KUKA KRL program: up24.src, up24.dat

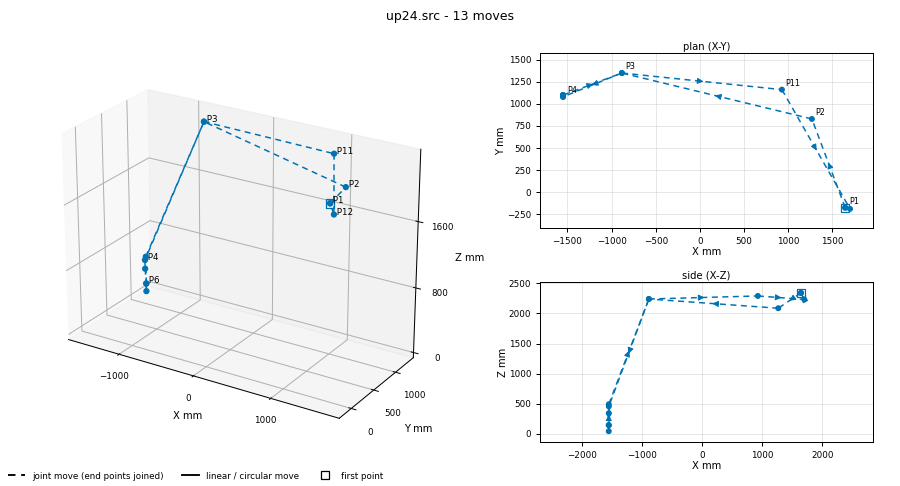
[picture p0: tool path of up24.src, 13 of 13 moves have a stored position in this frame; points joined in program order, loops and branches not executed]
--- up24.src ---
&ACCESS RV7
&REL 180
&COMMENT VW380 Ablegen AFO 115440
&PARAM DISKPATH = KRC:\R1\UPs
&PARAM TEMPLATE = C:\KRC\Roboter\Template\upvorgabe
&PARAM TPVW_VERSION = 8.1.8
&PARAM EDITMASK = Up999[1-999]
DEF UP24()
   ; FOLD UP Anfang;%{SE} %MKUKATPVW
   SPS_N=-1
   SPS_FERTIG=FALSE
   IF NOT CALLBYSELECT THEN
      INTERRUPT DECL 10 WHEN $CYCFLAG[254]==FALSE DO VW(#FB_STOP,TRUE)
      INTERRUPT ON 10
      INT10=TRUE
      VW_USR_R (#USR_INIT)
   ENDIF
   VW(#VW_INIT_UP,TRUE)
   ; ENDFOLD
   ;FOLD -- K2TUHR115425R01 -- ;%{PSE}%MKUKATPVW,%CVW_COM,%VCOMMENT,%P 1:Comment:, 2:K2TUHR115425R01
      ;FOLD {H}
         M_COMMENT("K2TUHR115425R01")
      ;ENDFOLD
   ;ENDFOLD
   ;FOLD -- VW370 Ablegen AFO 115440 -- ;%{PSE}%MKUKATPVW,%CVW_COM,%VCOMMENT,%P 1:Comment:, 2:VW370 Ablegen AFO 115440
      ;FOLD {H}
         M_COMMENT("VW370 Ablegen AFO 115440")
      ;ENDFOLD
   ;ENDFOLD
   ;FOLD -- Verriegelung (E43) an Rob 5440R01 EIN -- ;%{PSE}%MKUKATPVW,%CVW_COM,%VCOMMENT,%P 1:Comment:, 2:Verriegelung (E43) an Rob 5440R01 EIN
      ;FOLD {H}
         M_COMMENT("Verriegelung (E43) an Rob 5440R01 EIN")
      ;ENDFOLD
   ;ENDFOLD
   ;FOLD -- Verriegelung (E45) an Rob 5430R01 EIN -- ;%{PSE}%MKUKATPVW,%CVW_COM,%VCOMMENT,%P 1:Comment:, 2:Verriegelung (E45) an Rob 5430R01 EIN
      ;FOLD {H}
         M_COMMENT("Verriegelung (E45) an Rob 5430R01 EIN")
      ;ENDFOLD
   ;ENDFOLD
   ;FOLD -- Verriegelung (E54) an Rob 5450R01 EIN -- ;%{PSE}%MKUKATPVW,%CVW_COM,%VCOMMENT,%P 1:Comment:, 2:Verriegelung (E54) an Rob 5450R01 EIN
      ;FOLD {H}
         M_COMMENT("Verriegelung (E54) an Rob 5450R01 EIN")
      ;ENDFOLD
   ;ENDFOLD
   ;FOLD -- Profilfrei AFO 115440 AUS -- ;%{PSE}%MKUKATPVW,%CVW_COM,%VCOMMENT,%P 1:Comment:, 2:Profilfrei AFO 115440 AUS
      ;FOLD {H}
         M_COMMENT("Profilfrei AFO 115440 AUS")
      ;ENDFOLD
   ;ENDFOLD
   ;FOLD -- Profilfrei DT 115440 AUS -- ;%{PSE}%MKUKATPVW,%CVW_COM,%VCOMMENT,%P 1:Comment:, 2:Profilfrei DT 115440 AUS
      ;FOLD {H}
         M_COMMENT("Profilfrei DT 115440 AUS")
      ;ENDFOLD
   ;ENDFOLD
   ;FOLD -- Wartungsbereich -- ;%{PSE}%MKUKATPVW,%CVW_COM,%VCOMMENT,%P 1:Comment:, 2:Wartungsbereich
      ;FOLD {H}
         M_COMMENT("Wartungsbereich")
      ;ENDFOLD
   ;ENDFOLD
;FOLD PTP VB=100% VE=0% ACC=100% RobWzg=12 Base=0 SPSTrig=0[1/100s] P;%{P}%MKUKATPVW,%CMOVE8,%VPTP,%P 1:1, 2: VB=, 3:100, 4:%, 5: VE=, 6:0, 7:%, 8: ACC=, 9:100, 10:%, 11: RobWzg=, 12:12, 13: Base=, 14:0, 15: SPSTrig=, 16:0, 17:[1/100s], 18: P, 19:1, 20:-1, 21:1
;FOLD 1: FB PSPS = EIN;%{SE}%MKUKATPVW %CVW_SPS %VFBPSPS %P 2:FB PSPS = EIN,3: FBPSPS
;ENDFOLD
;FOLD 2: A23 = AUS;%{SE}%MKUKATPVW %CVW_SPS %VBOASG %P 2:A23 = AUS,3: BOASG
;ENDFOLD
;FOLD 3: t3 ( EIN ) = 0[1/10Sek];%{SE}%MKUKATPVW %CVW_SPS %VTASG %P 2:t3 ( EIN ) = 0[1/10Sek],3: TASG
;ENDFOLD
;FOLD 4: SPSMAKRO50 = EIN;%{SE}%MKUKATPVW %CVW_SPS %VMAKRO %P 2:SPSMAKRO50 = EIN,3: MAKRO
;ENDFOLD
;FOLD 5: SPSMAKRO53 = EIN;%{SE}%MKUKATPVW %CVW_SPS %VMAKRO %P 2:SPSMAKRO53 = EIN,3: MAKRO
;ENDFOLD
;FOLD 6: A42 = EIN;%{SE}%MKUKATPVW %CVW_SPS %VBOASG %P 2:A42 = EIN,3: BOASG
;ENDFOLD
;FOLD 7: A43 = EIN;%{SE}%MKUKATPVW %CVW_SPS %VBOASG %P 2:A43 = EIN,3: BOASG
;ENDFOLD
;FOLD 8: A44 = EIN;%{SE}%MKUKATPVW %CVW_SPS %VBOASG %P 2:A44 = EIN,3: BOASG
;ENDFOLD
;FOLD 9: A45 = EIN;%{SE}%MKUKATPVW %CVW_SPS %VBOASG %P 2:A45 = EIN,3: BOASG
;ENDFOLD
;FOLD 10: A47 = EIN;%{SE}%MKUKATPVW %CVW_SPS %VBOASG %P 2:A47 = EIN,3: BOASG
;ENDFOLD
;FOLD 11: A49 = EIN;%{SE}%MKUKATPVW %CVW_SPS %VBOASG %P 2:A49 = EIN,3: BOASG
;ENDFOLD
;FOLD 12: A50 = EIN;%{SE}%MKUKATPVW %CVW_SPS %VBOASG %P 2:A50 = EIN,3: BOASG
;ENDFOLD
;FOLD 13: A52 = EIN;%{SE}%MKUKATPVW %CVW_SPS %VBOASG %P 2:A52 = EIN,3: BOASG
;ENDFOLD
;FOLD 14: A54 = EIN;%{SE}%MKUKATPVW %CVW_SPS %VBOASG %P 2:A54 = EIN,3: BOASG
;ENDFOLD
;FOLD 15: A75 = EIN;%{SE}%MKUKATPVW %CVW_SPS %VBOASG %P 2:A75 = EIN,3: BOASG
;ENDFOLD
;FOLD 16: A76 = EIN;%{SE}%MKUKATPVW %CVW_SPS %VBOASG %P 2:A76 = EIN,3: BOASG
;ENDFOLD
;FOLD 17: A79 = EIN;%{SE}%MKUKATPVW %CVW_SPS %VBOASG %P 2:A79 = EIN,3: BOASG
;ENDFOLD
;FOLD 18: A80 = EIN;%{SE}%MKUKATPVW %CVW_SPS %VBOASG %P 2:A80 = EIN,3: BOASG
;ENDFOLD
;FOLD 19: A18 = EIN;%{SE}%MKUKATPVW %CVW_SPS %VBOASG %P 2:A18 = EIN,3: BOASG
;ENDFOLD
;FOLD 20: WARTE BIS E43 & E45 & E54 & !E59 & E60 & E75 & E76 & (!E18 + E19);%{SE}%MKUKATPVW %CVW_SPS %VWBOASG %P 2:WARTE BIS E43 & E45 & E54 & !E59 & E60 & E75 & E76 & (!E18 + E19),3: WBOASG
;ENDFOLD
;FOLD 21: A18 = AUS;%{SE}%MKUKATPVW %CVW_SPS %VBOASG %P 2:A18 = AUS,3: BOASG
;ENDFOLD
;FOLD 22: F2 = EIN;%{SE}%MKUKATPVW %CVW_SPS %VBOASG %P 2:F2 = EIN,3: BOASG
;ENDFOLD
;FOLD 23: SPSMAKRO343 = EIN;%{SE}%MKUKATPVW %CVW_SPS %VMAKRO %P 2:SPSMAKRO343 = EIN,3: MAKRO
;ENDFOLD
;FOLD 24: WARTE BIS M34;%{SE}%MKUKATPVW %CVW_SPS %VWBOASG %P 2:WARTE BIS M34,3: WBOASG
;ENDFOLD
;FOLD 25: A75 = AUS;%{SE}%MKUKATPVW %CVW_SPS %VBOASG %P 2:A75 = AUS,3: BOASG
;ENDFOLD
;FOLD 26: A76 = AUS;%{SE}%MKUKATPVW %CVW_SPS %VBOASG %P 2:A76 = AUS,3: BOASG
;ENDFOLD
;FOLD 27: A83 = EIN;%{SE}%MKUKATPVW %CVW_SPS %VBOASG %P 2:A83 = EIN,3: BOASG
;ENDFOLD
;FOLD 28: A85 = EIN;%{SE}%MKUKATPVW %CVW_SPS %VBOASG %P 2:A85 = EIN,3: BOASG
;ENDFOLD
;FOLD 29: A94 = EIN;%{SE}%MKUKATPVW %CVW_SPS %VBOASG %P 2:A94 = EIN,3: BOASG
;ENDFOLD
;FOLD 30: SPSMAKRO20 = EIN;%{SE}%MKUKATPVW %CVW_SPS %VMAKRO %P 2:SPSMAKRO20 = EIN,3: MAKRO
;ENDFOLD
;FOLD 31: WARTE BIS E23;%{SE}%MKUKATPVW %CVW_SPS %VWBOASG %P 2:WARTE BIS E23,3: WBOASG
;ENDFOLD
;FOLD 32: A23 = EIN;%{SE}%MKUKATPVW %CVW_SPS %VBOASG %P 2:A23 = EIN,3: BOASG
;ENDFOLD
;FOLD 33: FB PSPS = M1 & M28 & M30 & M32 & M34 & M78 & E60 & E75 & E76;%{SE}%MKUKATPVW %CVW_SPS %VFBPSPS %P 2:FB PSPS = M1 & M28 & M30 & M32 & M34 & M78 & E60 & E75 & E76,3: FBPSPS
;ENDFOLD
;FOLD {H}
VW_MPARA_ACT = P1_D
Act_P1 = P1
Act_P2 = P1
VW(#MPARA,TRUE)
SPS_FERTIG=FALSE
TRIGGER WHEN DISTANCE=1 DELAY=0 DO SPS_TRIG(1) PRIO=-1
PTP P1
$ADVANCE=1
WAIT FOR SPS_FERTIG
;ENDFOLD
;ENDFOLD
   ;FOLD PTP VB=100% VE=100% ACC=100% RobWzg=12 Base=0 SPSTrig=0[1/100s] P ;%{P}%MKUKATPVW,%CMOVE8,%VPTP,%P 1:1, 2: VB=, 3:100, 4:%, 5: VE=, 6:100, 7:%, 8: ACC=, 9:100, 10:%, 11: RobWzg=, 12:12, 13: Base=, 14:0, 15: SPSTrig=, 16:0, 17:[1/100s], 18: P, 19:2, 20:-1, 21:2
      ;FOLD 1: FB PSPS = M1 & M28 & M30 & M32 & M34 & M78 & E60 & E75 & E76 ;%{SE}%MKUKATPVW %CVW_SPS %VFBPSPS %P 2:FB PSPS = M1 & M28 & M30 & M32 & M34 & M78 & E60 & E75 & E76,3:FBPSPS
      ;ENDFOLD
      ;FOLD {H}
         VW_MPARA_ACT=P2_D
         Act_P1 = P2
         Act_P2 = P2
         VW(#MPARA,TRUE)
         SPS_FERTIG=FALSE
         TRIGGER WHEN DISTANCE=1 DELAY=0 DO SPS_TRIG(10002) PRIO=-1
         PTP P2 C_PTP C_VEL
         $ADVANCE=1
      ;ENDFOLD
   ;ENDFOLD
   ;FOLD PTP VB=100% VE=100% ACC=100% RobWzg=12 Base=0 SPSTrig=0[1/100s] P ;%{P}%MKUKATPVW,%CMOVE8,%VPTP,%P 1:1, 2: VB=, 3:100, 4:%, 5: VE=, 6:100, 7:%, 8: ACC=, 9:100, 10:%, 11: RobWzg=, 12:12, 13: Base=, 14:0, 15: SPSTrig=, 16:0, 17:[1/100s], 18: P, 19:3, 20:-1, 21:3
      ;FOLD 1: FB PSPS = M1 & M28 & M30 & M32 & M34 & M78 & E60 & E75 & E76 ;%{SE}%MKUKATPVW %CVW_SPS %VFBPSPS %P 2:FB PSPS = M1 & M28 & M30 & M32 & M34 & M78 & E60 & E75 & E76,3:FBPSPS
      ;ENDFOLD
      ;FOLD {H}
         VW_MPARA_ACT=P3_D
         Act_P1 = P3
         Act_P2 = P3
         VW(#MPARA,TRUE)
         SPS_FERTIG=FALSE
         TRIGGER WHEN DISTANCE=1 DELAY=0 DO SPS_TRIG(10003) PRIO=-1
         PTP P3 C_PTP C_VEL
         $ADVANCE=1
      ;ENDFOLD
   ;ENDFOLD
   ;FOLD PTP VB=100% VE=100% ACC=100% RobWzg=12 Base=0 SPSTrig=0[1/100s] P ;%{P}%MKUKATPVW,%CMOVE8,%VPTP,%P 1:1, 2: VB=, 3:100, 4:%, 5: VE=, 6:100, 7:%, 8: ACC=, 9:100, 10:%, 11: RobWzg=, 12:12, 13: Base=, 14:0, 15: SPSTrig=, 16:0, 17:[1/100s], 18: P, 19:4, 20:-1, 21:4
      ;FOLD 1: FB PSPS = M1 & M28 & M30 & M32 & M34 & M78 & E75 & E76 ;%{SE}%MKUKATPVW %CVW_SPS %VFBPSPS %P 2:FB PSPS = M1 & M28 & M30 & M32 & M34 & M78 & E75 & E76,3:FBPSPS
      ;ENDFOLD
      ;FOLD {H}
         VW_MPARA_ACT=P4_D
         Act_P1 = P4
         Act_P2 = P4
         VW(#MPARA,TRUE)
         SPS_FERTIG=FALSE
         TRIGGER WHEN DISTANCE=1 DELAY=0 DO SPS_TRIG(10004) PRIO=-1
         PTP P4 C_PTP C_VEL
         $ADVANCE=1
      ;ENDFOLD
   ;ENDFOLD
   ;FOLD PTP VB=100% VE=100% ACC=100% RobWzg=12 Base=0 SPSTrig=0[1/100s] P ;%{P}%MKUKATPVW,%CMOVE8,%VPTP,%P 1:1, 2: VB=, 3:100, 4:%, 5: VE=, 6:100, 7:%, 8: ACC=, 9:100, 10:%, 11: RobWzg=, 12:12, 13: Base=, 14:0, 15: SPSTrig=, 16:0, 17:[1/100s], 18: P, 19:5, 20:-1, 21:5
      ;FOLD 1: FB PSPS = M1 & M28 & M30 & M32 & M34 & M78 & E75 & E76 ;%{SE}%MKUKATPVW %CVW_SPS %VFBPSPS %P 2:FB PSPS = M1 & M28 & M30 & M32 & M34 & M78 & E75 & E76,3:FBPSPS
      ;ENDFOLD
      ;FOLD {H}
         VW_MPARA_ACT=P5_D
         Act_P1 = P5
         Act_P2 = P5
         VW(#MPARA,TRUE)
         SPS_FERTIG=FALSE
         TRIGGER WHEN DISTANCE=1 DELAY=0 DO SPS_TRIG(10005) PRIO=-1
         PTP P5 C_PTP C_VEL
         $ADVANCE=1
      ;ENDFOLD
   ;ENDFOLD
   ;FOLD PTP VB=100% VE=10% ACC=100% RobWzg=12 Base=0 SPSTrig=0[1/100s] P ;%{P}%MKUKATPVW,%CMOVE8,%VPTP,%P 1:1, 2: VB=, 3:100, 4:%, 5: VE=, 6:10, 7:%, 8: ACC=, 9:100, 10:%, 11: RobWzg=, 12:12, 13: Base=, 14:0, 15: SPSTrig=, 16:0, 17:[1/100s], 18: P, 19:6, 20:-1, 21:6
      ;FOLD 1: FB PSPS = M1 & M28 & M30 & M32 & M34 & M78 & E75 & E76 ;%{SE}%MKUKATPVW %CVW_SPS %VFBPSPS %P 2:FB PSPS = M1 & M28 & M30 & M32 & M34 & M78 & E75 & E76,3:FBPSPS
      ;ENDFOLD
      ;FOLD {H}
         VW_MPARA_ACT=P6_D
         Act_P1 = P6
         Act_P2 = P6
         VW(#MPARA,TRUE)
         SPS_FERTIG=FALSE
         TRIGGER WHEN DISTANCE=1 DELAY=0 DO SPS_TRIG(10006) PRIO=-1
         PTP P6 C_PTP C_VEL
         $ADVANCE=1
      ;ENDFOLD
   ;ENDFOLD
   ;FOLD -- Bauteil ablegen AFO 115440 -- ;%{PSE}%MKUKATPVW,%CVW_COM,%VCOMMENT,%P 1:Comment:, 2:Bauteil ablegen AFO 115440
      ;FOLD {H}
         M_COMMENT("Bauteil ablegen AFO 115440")
      ;ENDFOLD
   ;ENDFOLD
   ;FOLD -- Greifer auf -- ;%{PSE}%MKUKATPVW,%CVW_COM,%VCOMMENT,%P 1:Comment:, 2:Greifer auf
      ;FOLD {H}
         M_COMMENT("Greifer auf")
      ;ENDFOLD
   ;ENDFOLD
   ;FOLD LIN VB=250[mm/s] VE=0% ACC=100% RobWzg=12 Base=0 SPSTrig=5[1/100s] P ;%{P}%MKUKATPVW,%CMOVE8,%VLIN,%P 1:2, 2: VB=, 3:250, 4:[mm/s], 5: VE=, 6:0, 7:%, 8: ACC=, 9:100, 10:%, 11: RobWzg=, 12:12, 13: Base=, 14:0, 15: SPSTrig=, 16:5, 17:[1/100s], 18: P, 19:7, 20:-1, 21:7
      ;FOLD 1: FB PSPS = EIN ;%{SE}%MKUKATPVW %CVW_SPS %VFBPSPS %P 2:FB PSPS = EIN,3:FBPSPS
      ;ENDFOLD
      ;FOLD 2: A23 = AUS ;%{SE}%MKUKATPVW %CVW_SPS %VBOASG %P 2:A23 = AUS,3:BOASG
      ;ENDFOLD
      ;FOLD 3: A73 = EIN ;%{SE}%MKUKATPVW %CVW_SPS %VBOASG %P 2:A73 = EIN,3:BOASG
      ;ENDFOLD
      ;FOLD 4: WARTE BIS E59 & !E60 ;%{SE}%MKUKATPVW %CVW_SPS %VWBOASG %P 2:WARTE BIS E59 & !E60,3:WBOASG
      ;ENDFOLD
      ;FOLD 5: A74 = EIN ;%{SE}%MKUKATPVW %CVW_SPS %VBOASG %P 2:A74 = EIN,3:BOASG
      ;ENDFOLD
      ;FOLD 6: F1 = EIN ;%{SE}%MKUKATPVW %CVW_SPS %VBOASG %P 2:F1 = EIN,3:BOASG
      ;ENDFOLD
      ;FOLD 7: SPSMAKRO342 = EIN ;%{SE}%MKUKATPVW %CVW_SPS %VMAKRO %P 2:SPSMAKRO342 = EIN,3:MAKRO
      ;ENDFOLD
      ;FOLD 8: SPSMAKRO340 = EIN ;%{SE}%MKUKATPVW %CVW_SPS %VMAKRO %P 2:SPSMAKRO340 = EIN,3:MAKRO
      ;ENDFOLD
      ;FOLD 9: WARTE BIS M31 & M34 ;%{SE}%MKUKATPVW %CVW_SPS %VWBOASG %P 2:WARTE BIS M31 & M34,3:WBOASG
      ;ENDFOLD
      ;FOLD 10: SPSMAKRO4 = EIN ;%{SE}%MKUKATPVW %CVW_SPS %VMAKRO %P 2:SPSMAKRO4 = EIN,3:MAKRO
      ;ENDFOLD
      ;FOLD 11: WARTE BIS E74 ;%{SE}%MKUKATPVW %CVW_SPS %VWBOASG %P 2:WARTE BIS E74,3:WBOASG
      ;ENDFOLD
      ;FOLD 12: A73 = AUS ;%{SE}%MKUKATPVW %CVW_SPS %VBOASG %P 2:A73 = AUS,3:BOASG
      ;ENDFOLD
      ;FOLD 13: A74 = AUS ;%{SE}%MKUKATPVW %CVW_SPS %VBOASG %P 2:A74 = AUS,3:BOASG
      ;ENDFOLD
      ;FOLD 14: WARTE BIS E23 ;%{SE}%MKUKATPVW %CVW_SPS %VWBOASG %P 2:WARTE BIS E23,3:WBOASG
      ;ENDFOLD
      ;FOLD 15: A23 = EIN ;%{SE}%MKUKATPVW %CVW_SPS %VBOASG %P 2:A23 = EIN,3:BOASG
      ;ENDFOLD
      ;FOLD 16: FB PSPS = M28 & M30 & M31 & M34 & M78 & E59 & E74 & E76 ;%{SE}%MKUKATPVW %CVW_SPS %VFBPSPS %P 2:FB PSPS = M28 & M30 & M31 & M34 & M78 & E59 & E74 & E76,3:FBPSPS
      ;ENDFOLD
      ;FOLD {H}
         VW_MPARA_ACT=P7_D
         Act_P1 = P7
         Act_P2 = P7
         VW(#MPARA,TRUE)
         SPS_FERTIG=FALSE
         TRIGGER WHEN DISTANCE=1 DELAY=-50 DO SPS_TRIG(7) PRIO=-1
         LIN P7
         $ADVANCE=1
         WAIT FOR SPS_FERTIG
      ;ENDFOLD
   ;ENDFOLD
   ;FOLD LIN VB=300[mm/s] VE=100% ACC=100% RobWzg=12 Base=0 SPSTrig=0[1/100s] P ;%{P}%MKUKATPVW,%CMOVE8,%VLIN,%P 1:2, 2: VB=, 3:300, 4:[mm/s], 5: VE=, 6:100, 7:%, 8: ACC=, 9:100, 10:%, 11: RobWzg=, 12:12, 13: Base=, 14:0, 15: SPSTrig=, 16:0, 17:[1/100s], 18: P, 19:8, 20:-1, 21:8
      ;FOLD 1: FB PSPS = M13 & M28 & M30 & M31 & M34 & M78 & E59 & E74 & E76 ;%{SE}%MKUKATPVW %CVW_SPS %VFBPSPS %P 2:FB PSPS = M13 & M28 & M30 & M31 & M34 & M78 & E59 & E74 & E76,3:FBPSPS
      ;ENDFOLD
      ;FOLD {H}
         VW_MPARA_ACT=P8_D
         Act_P1 = P8
         Act_P2 = P8
         VW(#MPARA,TRUE)
         SPS_FERTIG=FALSE
         TRIGGER WHEN DISTANCE=1 DELAY=0 DO SPS_TRIG(10008) PRIO=-1
         LIN P8 C_VEL
         $ADVANCE=1
      ;ENDFOLD
   ;ENDFOLD
   ;FOLD PTP VB=100% VE=100% ACC=100% RobWzg=12 Base=0 SPSTrig=0[1/100s] P ;%{P}%MKUKATPVW,%CMOVE8,%VPTP,%P 1:1, 2: VB=, 3:100, 4:%, 5: VE=, 6:100, 7:%, 8: ACC=, 9:100, 10:%, 11: RobWzg=, 12:12, 13: Base=, 14:0, 15: SPSTrig=, 16:0, 17:[1/100s], 18: P, 19:9, 20:-1, 21:9
      ;FOLD 1: FB PSPS = M13 & M28 & M30 & M31 & M34 & M78 & E59 & E74 & E76 ;%{SE}%MKUKATPVW %CVW_SPS %VFBPSPS %P 2:FB PSPS = M13 & M28 & M30 & M31 & M34 & M78 & E59 & E74 & E76,3:FBPSPS
      ;ENDFOLD
      ;FOLD {H}
         VW_MPARA_ACT=P9_D
         Act_P1 = P9
         Act_P2 = P9
         VW(#MPARA,TRUE)
         SPS_FERTIG=FALSE
         TRIGGER WHEN DISTANCE=1 DELAY=0 DO SPS_TRIG(10009) PRIO=-1
         PTP P9 C_PTP C_VEL
         $ADVANCE=1
      ;ENDFOLD
   ;ENDFOLD
   ;FOLD -- Profilfrei AFO 115440 EIN -- ;%{PSE}%MKUKATPVW,%CVW_COM,%VCOMMENT,%P 1:Comment:, 2:Profilfrei AFO 115440 EIN
      ;FOLD {H}
         M_COMMENT("Profilfrei AFO 115440 EIN")
      ;ENDFOLD
   ;ENDFOLD
   ;FOLD -- Verriegelung (E45) an Rob 5430R01 AUS -- ;%{PSE}%MKUKATPVW,%CVW_COM,%VCOMMENT,%P 1:Comment:, 2:Verriegelung (E45) an Rob 5430R01 AUS
      ;FOLD {H}
         M_COMMENT("Verriegelung (E45) an Rob 5430R01 AUS")
      ;ENDFOLD
   ;ENDFOLD
;FOLD PTP VB=100% VE=100% ACC=100% RobWzg=12 Base=0 SPSTrig=0[1/100s] P;%{P}%MKUKATPVW,%CMOVE8,%VPTP,%P 1:1, 2: VB=, 3:100, 4:%, 5: VE=, 6:100, 7:%, 8: ACC=, 9:100, 10:%, 11: RobWzg=, 12:12, 13: Base=, 14:0, 15: SPSTrig=, 16:0, 17:[1/100s], 18: P, 19:10, 20:-1, 21:10
;FOLD 1: FB PSPS = EIN;%{SE}%MKUKATPVW %CVW_SPS %VFBPSPS %P 2:FB PSPS = EIN,3: FBPSPS
;ENDFOLD
;FOLD 2: A75 = EIN;%{SE}%MKUKATPVW %CVW_SPS %VBOASG %P 2:A75 = EIN,3: BOASG
;ENDFOLD
;FOLD 3: A45 = EIN;%{SE}%MKUKATPVW %CVW_SPS %VBOASG %P 2:A45 = EIN,3: BOASG
;ENDFOLD
;FOLD 4: FB PSPS = M13 & M30 & M31 & M34 & M78 & E43 & E54 & E76;%{SE}%MKUKATPVW %CVW_SPS %VFBPSPS %P 2:FB PSPS = M13 & M30 & M31 & M34 & M78 & E43 & E54 & E76,3: FBPSPS
;ENDFOLD
;FOLD {H}
VW_MPARA_ACT = P10_D
Act_P1 = P10
Act_P2 = P10
VW(#MPARA,TRUE)
SPS_FERTIG=FALSE
TRIGGER WHEN DISTANCE=1 DELAY=0 DO SPS_TRIG(10010) PRIO=-1
PTP P10 C_PTP C_VEL
$ADVANCE=1
;ENDFOLD
;ENDFOLD
   ;FOLD -- Verriegelung (E43) an Rob 5440R01 AUS -- ;%{PSE}%MKUKATPVW,%CVW_COM,%VCOMMENT,%P 1:Comment:, 2:Verriegelung (E43) an Rob 5440R01 AUS
      ;FOLD {H}
         M_COMMENT("Verriegelung (E43) an Rob 5440R01 AUS")
      ;ENDFOLD
   ;ENDFOLD
   ;FOLD -- Verriegelung (E54) an Rob 5450R01 AUS -- ;%{PSE}%MKUKATPVW,%CVW_COM,%VCOMMENT,%P 1:Comment:, 2:Verriegelung (E54) an Rob 5450R01 AUS
      ;FOLD {H}
         M_COMMENT("Verriegelung (E54) an Rob 5450R01 AUS")
      ;ENDFOLD
   ;ENDFOLD
;FOLD PTP VB=100% VE=100% ACC=100% RobWzg=12 Base=0 SPSTrig=0[1/100s] P;%{P}%MKUKATPVW,%CMOVE8,%VPTP,%P 1:1, 2: VB=, 3:100, 4:%, 5: VE=, 6:100, 7:%, 8: ACC=, 9:100, 10:%, 11: RobWzg=, 12:12, 13: Base=, 14:0, 15: SPSTrig=, 16:0, 17:[1/100s], 18: P, 19:11, 20:-1, 21:11
;FOLD 1: FB PSPS = EIN;%{SE}%MKUKATPVW %CVW_SPS %VFBPSPS %P 2:FB PSPS = EIN,3: FBPSPS
;ENDFOLD
;FOLD 2: A43 = EIN;%{SE}%MKUKATPVW %CVW_SPS %VBOASG %P 2:A43 = EIN,3: BOASG
;ENDFOLD
;FOLD 3: A54 = EIN;%{SE}%MKUKATPVW %CVW_SPS %VBOASG %P 2:A54 = EIN,3: BOASG
;ENDFOLD
;FOLD 4: FB PSPS = M13 & M30 & M31 & M34 & M78 & E76;%{SE}%MKUKATPVW %CVW_SPS %VFBPSPS %P 2:FB PSPS = M13 & M30 & M31 & M34 & M78 & E76,3: FBPSPS
;ENDFOLD
;FOLD {H}
VW_MPARA_ACT = P11_D
Act_P1 = P11
Act_P2 = P11
VW(#MPARA,TRUE)
SPS_FERTIG=FALSE
TRIGGER WHEN DISTANCE=1 DELAY=0 DO SPS_TRIG(10011) PRIO=-1
PTP P11 C_PTP C_VEL
$ADVANCE=1
;ENDFOLD
;ENDFOLD
   ;FOLD PTP VB=100% VE=100% ACC=100% RobWzg=12 Base=0 SPSTrig=0[1/100s] P ;%{P}%MKUKATPVW,%CMOVE8,%VPTP,%P 1:1, 2: VB=, 3:100, 4:%, 5: VE=, 6:100, 7:%, 8: ACC=, 9:100, 10:%, 11: RobWzg=, 12:12, 13: Base=, 14:0, 15: SPSTrig=, 16:0, 17:[1/100s], 18: P, 19:12, 20:-1, 21:12
      ;FOLD 1: FB PSPS = M13 & M30 & M31 & M34 & M78 & E76 ;%{SE}%MKUKATPVW %CVW_SPS %VFBPSPS %P 2:FB PSPS = M13 & M30 & M31 & M34 & M78 & E76,3:FBPSPS
      ;ENDFOLD
      ;FOLD {H}
         VW_MPARA_ACT=P12_D
         Act_P1 = P12
         Act_P2 = P12
         VW(#MPARA,TRUE)
         SPS_FERTIG=FALSE
         TRIGGER WHEN DISTANCE=1 DELAY=0 DO SPS_TRIG(10012) PRIO=-1
         PTP P12 C_PTP C_VEL
         $ADVANCE=1
      ;ENDFOLD
   ;ENDFOLD
   ;FOLD -- Profilfrei DT 115440 EIN -- ;%{PSE}%MKUKATPVW,%CVW_COM,%VCOMMENT,%P 1:Comment:, 2:Profilfrei DT 115440 EIN
      ;FOLD {H}
         M_COMMENT("Profilfrei DT 115440 EIN")
      ;ENDFOLD
   ;ENDFOLD
   ;FOLD PTP VB=100% VE=0% ACC=100% RobWzg=12 Base=0 SPSTrig=0[1/100s] P ;%{P}%MKUKATPVW,%CMOVE8,%VPTP,%P 1:1, 2: VB=, 3:100, 4:%, 5: VE=, 6:0, 7:%, 8: ACC=, 9:100, 10:%, 11: RobWzg=, 12:12, 13: Base=, 14:0, 15: SPSTrig=, 16:0, 17:[1/100s], 18: P, 19:13, 20:-1, 21:13
      ;FOLD 1: FB PSPS = EIN ;%{SE}%MKUKATPVW %CVW_SPS %VFBPSPS %P 2:FB PSPS = EIN,3:FBPSPS
      ;ENDFOLD
      ;FOLD 2: A23 = AUS ;%{SE}%MKUKATPVW %CVW_SPS %VBOASG %P 2:A23 = AUS,3:BOASG
      ;ENDFOLD
      ;FOLD 3: A76 = EIN ;%{SE}%MKUKATPVW %CVW_SPS %VBOASG %P 2:A76 = EIN,3:BOASG
      ;ENDFOLD
      ;FOLD 4: t3 ( EIN ) = STOP ;%{SE}%MKUKATPVW %CVW_SPS %VTSTOP %P 2:t3 ( EIN ) = STOP,3:TSTOP
      ;ENDFOLD
      ;FOLD 5: WARTE BIS E23 ;%{SE}%MKUKATPVW %CVW_SPS %VWBOASG %P 2:WARTE BIS E23,3:WBOASG
      ;ENDFOLD
      ;FOLD 6: A23 = EIN ;%{SE}%MKUKATPVW %CVW_SPS %VBOASG %P 2:A23 = EIN,3:BOASG
      ;ENDFOLD
      ;FOLD 7: FB PSPS = M13 & M30 & M31 & M34 & M78 ;%{SE}%MKUKATPVW %CVW_SPS %VFBPSPS %P 2:FB PSPS = M13 & M30 & M31 & M34 & M78,3:FBPSPS
      ;ENDFOLD
      ;FOLD {H}
         VW_MPARA_ACT=P13_D
         Act_P1 = P13
         Act_P2 = P13
         VW(#MPARA,TRUE)
         SPS_FERTIG=FALSE
         TRIGGER WHEN DISTANCE=1 DELAY=0 DO SPS_TRIG(13) PRIO=-1
         PTP P13
         $ADVANCE=1
         WAIT FOR SPS_FERTIG
      ;ENDFOLD
   ;ENDFOLD
   ; FOLD ;%{H}
END
DEF SPS_TRIG(NO :IN)
   INT NO
   INT VW_STOP
   BOOL UES
   VW_STOP=$VW_PSPS_STOP
   IF NO>10000 THEN
      NO=NO-10000
      UES=TRUE
   ELSE
      UES=FALSE
   ENDIF
   ; FOLD ;%{H}
   IF ((VW_STOP B_AND 'B0001') > 0) THEN
      ;-- Trigger vorzeitig geschaltet (delay < 0) oder MStep
      IF (((VW_STOP B_AND 'B0110') > 0) AND ($MODE_OP<>#EX)) THEN
         ;-- MStep oder BCO Bewegung
         HALT
      ENDIF
   ENDIF
   ; ENDFOLD
   IF (SEARCH_END) THEN
      SEARCH_END = FALSE
      INTERRUPT OFF 39
   ENDIF
   SWITCH NO
      CASE 1
;FOLD SPS_TRIG1 {H}
VALCYCFL30=$CYCFLAG[254]
$CYCFLAG[254]=(TRUE) AND $CYCFLAG[255] OR ($TIMER[61]<0)
VW(#FB_CHECK,TRUE)
$OUT[23]=FALSE
VW(#SET_TIME,TRUE,3,0,0)
SEL_RES=SELECT(#MAKRO,50,TRUE,,,,,FALSE)
SEL_RES=SELECT(#MAKRO,53,TRUE,,,,,FALSE)
$OUT[42]=TRUE
$OUT[43]=TRUE
$OUT[44]=TRUE
$OUT[45]=TRUE
$OUT[47]=TRUE
$OUT[49]=TRUE
$OUT[50]=TRUE
$OUT[52]=TRUE
$OUT[54]=TRUE
$OUT[75]=TRUE
$OUT[76]=TRUE
$OUT[79]=TRUE
$OUT[80]=TRUE
$OUT[18]=TRUE
$LOOP_MSG[]="E43 & E45 & E54 & !E59 & E60 & E75 & E76 & (!E18 + E19)"
$LOOP_CONT=TRUE
WAIT FOR ($IN[43] AND $IN[45] AND $IN[54] AND NOT $IN[59] AND $IN[60] AND $IN[75] AND $IN[76] AND (NOT $IN[18] OR $IN[19])) OR (NOT $LOOP_CONT AND ($MODE_OP<>#EX))
$LOOP_MSG[]="                                                                                                                                "
$OUT[18]=FALSE
$FLAG[2]=TRUE
SEL_RES=SELECT(#MAKRO,343,TRUE,,,,,FALSE)
$LOOP_MSG[]="M34"
$LOOP_CONT=TRUE
WAIT FOR ($CYCFLAG[34]) OR (NOT $LOOP_CONT AND ($MODE_OP<>#EX))
$LOOP_MSG[]="                                                                                                                                "
$OUT[75]=FALSE
$OUT[76]=FALSE
$OUT[83]=TRUE
$OUT[85]=TRUE
$OUT[94]=TRUE
SEL_RES=SELECT(#MAKRO,20,TRUE,,,,,FALSE)
$LOOP_MSG[]="E23"
$LOOP_CONT=TRUE
WAIT FOR ($IN[23]) OR (NOT $LOOP_CONT AND ($MODE_OP<>#EX))
$LOOP_MSG[]="                                                                                                                                "
$OUT[23]=TRUE
VALCYCFL30=$CYCFLAG[254]
$CYCFLAG[254]=($CYCFLAG[1] AND $CYCFLAG[28] AND $CYCFLAG[30] AND $CYCFLAG[32] AND $CYCFLAG[34] AND $CYCFLAG[78] AND $IN[60] AND $IN[75] AND $IN[76]) AND $CYCFLAG[255] OR ($TIMER[61]<0)
VW(#FB_CHECK,TRUE)
;ENDFOLD
      CASE 2
         ;FOLD SPS_TRIG2{H}
            VALCYCFL30=$CYCFLAG[254]
            $CYCFLAG[254]=($CYCFLAG[1] AND $CYCFLAG[28] AND $CYCFLAG[30] AND $CYCFLAG[32] AND $CYCFLAG[34] AND $CYCFLAG[78] AND $IN[60] AND $IN[75] AND $IN[76]) AND $CYCFLAG[255] OR ($TIMER[61]<0)
            VW(#FB_CHECK,TRUE)
         ;ENDFOLD
      CASE 3
         ;FOLD SPS_TRIG3{H}
            VALCYCFL30=$CYCFLAG[254]
            $CYCFLAG[254]=($CYCFLAG[1] AND $CYCFLAG[28] AND $CYCFLAG[30] AND $CYCFLAG[32] AND $CYCFLAG[34] AND $CYCFLAG[78] AND $IN[60] AND $IN[75] AND $IN[76]) AND $CYCFLAG[255] OR ($TIMER[61]<0)
            VW(#FB_CHECK,TRUE)
         ;ENDFOLD
      CASE 4
         ;FOLD SPS_TRIG4{H}
            VALCYCFL30=$CYCFLAG[254]
            $CYCFLAG[254]=($CYCFLAG[1] AND $CYCFLAG[28] AND $CYCFLAG[30] AND $CYCFLAG[32] AND $CYCFLAG[34] AND $CYCFLAG[78] AND $IN[75] AND $IN[76]) AND $CYCFLAG[255] OR ($TIMER[61]<0)
            VW(#FB_CHECK,TRUE)
         ;ENDFOLD
      CASE 5
         ;FOLD SPS_TRIG5{H}
            VALCYCFL30=$CYCFLAG[254]
            $CYCFLAG[254]=($CYCFLAG[1] AND $CYCFLAG[28] AND $CYCFLAG[30] AND $CYCFLAG[32] AND $CYCFLAG[34] AND $CYCFLAG[78] AND $IN[75] AND $IN[76]) AND $CYCFLAG[255] OR ($TIMER[61]<0)
            VW(#FB_CHECK,TRUE)
         ;ENDFOLD
      CASE 6
         ;FOLD SPS_TRIG6{H}
            VALCYCFL30=$CYCFLAG[254]
            $CYCFLAG[254]=($CYCFLAG[1] AND $CYCFLAG[28] AND $CYCFLAG[30] AND $CYCFLAG[32] AND $CYCFLAG[34] AND $CYCFLAG[78] AND $IN[75] AND $IN[76]) AND $CYCFLAG[255] OR ($TIMER[61]<0)
            VW(#FB_CHECK,TRUE)
         ;ENDFOLD
      CASE 7
         ;FOLD SPS_TRIG7{H}
            VALCYCFL30=$CYCFLAG[254]
            $CYCFLAG[254]=(TRUE) AND $CYCFLAG[255] OR ($TIMER[61]<0)
            VW(#FB_CHECK,TRUE)
            $OUT[23] = FALSE
            $OUT[73] = TRUE
            $LOOP_MSG[]="E59 & !E60"
            $LOOP_CONT=TRUE
            WAIT FOR ($IN[59] AND NOT $IN[60]) OR (NOT $LOOP_CONT AND ($MODE_OP<>#EX))
            $LOOP_MSG[]="                                                                                                                                "
            $OUT[74] = TRUE
            $FLAG[1] = TRUE
            SEL_RES=SELECT(#MAKRO,342,TRUE,,,,,FALSE)
            SEL_RES=SELECT(#MAKRO,340,TRUE,,,,,FALSE)
            $LOOP_MSG[]="M31 & M34"
            $LOOP_CONT=TRUE
            WAIT FOR ($CYCFLAG[31] AND $CYCFLAG[34]) OR (NOT $LOOP_CONT AND ($MODE_OP<>#EX))
            $LOOP_MSG[]="                                                                                                                                "
            SEL_RES=SELECT(#MAKRO,4,TRUE,,,,,FALSE)
            $LOOP_MSG[]="E74"
            $LOOP_CONT=TRUE
            WAIT FOR ($IN[74]) OR (NOT $LOOP_CONT AND ($MODE_OP<>#EX))
            $LOOP_MSG[]="                                                                                                                                "
            $OUT[73] = FALSE
            $OUT[74] = FALSE
            $LOOP_MSG[]="E23"
            $LOOP_CONT=TRUE
            WAIT FOR ($IN[23]) OR (NOT $LOOP_CONT AND ($MODE_OP<>#EX))
            $LOOP_MSG[]="                                                                                                                                "
            $OUT[23] = TRUE
            VALCYCFL30=$CYCFLAG[254]
            $CYCFLAG[254]=($CYCFLAG[28] AND $CYCFLAG[30] AND $CYCFLAG[31] AND $CYCFLAG[34] AND $CYCFLAG[78] AND $IN[59] AND $IN[74] AND $IN[76]) AND $CYCFLAG[255] OR ($TIMER[61]<0)
            VW(#FB_CHECK,TRUE)
         ;ENDFOLD
      CASE 8
         ;FOLD SPS_TRIG8{H}
            VALCYCFL30=$CYCFLAG[254]
            $CYCFLAG[254]=($CYCFLAG[13] AND $CYCFLAG[28] AND $CYCFLAG[30] AND $CYCFLAG[31] AND $CYCFLAG[34] AND $CYCFLAG[78] AND $IN[59] AND $IN[74] AND $IN[76]) AND $CYCFLAG[255] OR ($TIMER[61]<0)
            VW(#FB_CHECK,TRUE)
         ;ENDFOLD
      CASE 9
         ;FOLD SPS_TRIG9{H}
            VALCYCFL30=$CYCFLAG[254]
            $CYCFLAG[254]=($CYCFLAG[13] AND $CYCFLAG[28] AND $CYCFLAG[30] AND $CYCFLAG[31] AND $CYCFLAG[34] AND $CYCFLAG[78] AND $IN[59] AND $IN[74] AND $IN[76]) AND $CYCFLAG[255] OR ($TIMER[61]<0)
            VW(#FB_CHECK,TRUE)
         ;ENDFOLD
      CASE 10
;FOLD SPS_TRIG10 {H}
VALCYCFL30=$CYCFLAG[254]
$CYCFLAG[254]=(TRUE) AND $CYCFLAG[255] OR ($TIMER[61]<0)
VW(#FB_CHECK,TRUE)
$OUT[75]=TRUE
$OUT[45]=TRUE
VALCYCFL30=$CYCFLAG[254]
$CYCFLAG[254]=($CYCFLAG[13] AND $CYCFLAG[30] AND $CYCFLAG[31] AND $CYCFLAG[34] AND $CYCFLAG[78] AND $IN[43] AND $IN[54] AND $IN[76]) AND $CYCFLAG[255] OR ($TIMER[61]<0)
VW(#FB_CHECK,TRUE)
;ENDFOLD
      CASE 11
;FOLD SPS_TRIG11 {H}
VALCYCFL30=$CYCFLAG[254]
$CYCFLAG[254]=(TRUE) AND $CYCFLAG[255] OR ($TIMER[61]<0)
VW(#FB_CHECK,TRUE)
$OUT[43]=TRUE
$OUT[54]=TRUE
VALCYCFL30=$CYCFLAG[254]
$CYCFLAG[254]=($CYCFLAG[13] AND $CYCFLAG[30] AND $CYCFLAG[31] AND $CYCFLAG[34] AND $CYCFLAG[78] AND $IN[76]) AND $CYCFLAG[255] OR ($TIMER[61]<0)
VW(#FB_CHECK,TRUE)
;ENDFOLD
      CASE 12
         ;FOLD SPS_TRIG12{H}
            VALCYCFL30=$CYCFLAG[254]
            $CYCFLAG[254]=($CYCFLAG[13] AND $CYCFLAG[30] AND $CYCFLAG[31] AND $CYCFLAG[34] AND $CYCFLAG[78] AND $IN[76]) AND $CYCFLAG[255] OR ($TIMER[61]<0)
            VW(#FB_CHECK,TRUE)
         ;ENDFOLD
      CASE 13
         ;FOLD SPS_TRIG13{H}
            VALCYCFL30=$CYCFLAG[254]
            $CYCFLAG[254]=(TRUE) AND $CYCFLAG[255] OR ($TIMER[61]<0)
            VW(#FB_CHECK,TRUE)
            $OUT[23] = FALSE
            $OUT[76] = TRUE
            VW(#SET_TIME,TRUE,3,1,0)
            $LOOP_MSG[]="E23"
            $LOOP_CONT=TRUE
            WAIT FOR ($IN[23]) OR (NOT $LOOP_CONT AND ($MODE_OP<>#EX))
            $LOOP_MSG[]="                                                                                                                                "
            $OUT[23] = TRUE
            VALCYCFL30=$CYCFLAG[254]
            $CYCFLAG[254]=($CYCFLAG[13] AND $CYCFLAG[30] AND $CYCFLAG[31] AND $CYCFLAG[34] AND $CYCFLAG[78]) AND $CYCFLAG[255] OR ($TIMER[61]<0)
            VW(#FB_CHECK,TRUE)
         ;ENDFOLD
      CASE 14
         ;FOLD SPS_TRIG14{H}
         ;ENDFOLD
      CASE 15
         ;FOLD SPS_TRIG15{H}
         ;ENDFOLD
      CASE 16
         ;FOLD SPS_TRIG16{H}
         ;ENDFOLD
      CASE 17
         ;FOLD SPS_TRIG17{H}
         ;ENDFOLD
      CASE 18
         ;FOLD SPS_TRIG18{H}
         ;ENDFOLD
      CASE 19
         ;FOLD SPS_TRIG19{H}
         ;ENDFOLD
      CASE 20
         ;FOLD SPS_TRIG20{H}
         ;ENDFOLD
      CASE 21
         ;FOLD SPS_TRIG21{H}
         ;ENDFOLD
      CASE 22
         ;FOLD SPS_TRIG22{H}
         ;ENDFOLD
      CASE 23
         ;FOLD SPS_TRIG23{H}
         ;ENDFOLD
      CASE 24
         ;FOLD SPS_TRIG24{H}
         ;ENDFOLD
      CASE 25
         ;FOLD SPS_TRIG25{H}
         ;ENDFOLD
      CASE 26
         ;FOLD SPS_TRIG26{H}
         ;ENDFOLD
      CASE 27
         ;FOLD SPS_TRIG27{H}
         ;ENDFOLD
      CASE 28
         ;FOLD SPS_TRIG28{H}
         ;ENDFOLD
      CASE 29
         ;FOLD SPS_TRIG29{H}
         ;ENDFOLD
      CASE 30
         ;FOLD SPS_TRIG30{H}
         ;ENDFOLD
      CASE 31
         ;FOLD SPS_TRIG31{H}
         ;ENDFOLD
      CASE 32
         ;FOLD SPS_TRIG32{H}
         ;ENDFOLD
      CASE 33
         ;FOLD SPS_TRIG33{H}
         ;ENDFOLD
      CASE 34
         ;FOLD SPS_TRIG34{H}
         ;ENDFOLD
      CASE 35
         ;FOLD SPS_TRIG35{H}
         ;ENDFOLD
      CASE 36
         ;FOLD SPS_TRIG36{H}
         ;ENDFOLD
      CASE 37
         ;FOLD SPS_TRIG37{H}
         ;ENDFOLD
      CASE 38
         ;FOLD SPS_TRIG38{H}
         ;ENDFOLD
      CASE 39
         ;FOLD SPS_TRIG39{H}
         ;ENDFOLD
      CASE 40
         ;FOLD SPS_TRIG40{H}
         ;ENDFOLD
      CASE 41
         ;FOLD SPS_TRIG41{H}
         ;ENDFOLD
      CASE 42
         ;FOLD SPS_TRIG42{H}
         ;ENDFOLD
      CASE 43
         ;FOLD SPS_TRIG43{H}
         ;ENDFOLD
      CASE 44
         ;FOLD SPS_TRIG44{H}
         ;ENDFOLD
      CASE 45
         ;FOLD SPS_TRIG45{H}
         ;ENDFOLD
      CASE 46
         ;FOLD SPS_TRIG46{H}
         ;ENDFOLD
      CASE 47
         ;FOLD SPS_TRIG47{H}
         ;ENDFOLD
      CASE 48
         ;FOLD SPS_TRIG48{H}
         ;ENDFOLD
      CASE 49
         ;FOLD SPS_TRIG49{H}
         ;ENDFOLD
      CASE 50
         ;FOLD SPS_TRIG50{H}
         ;ENDFOLD
      CASE 51
         ;FOLD SPS_TRIG51{H}
         ;ENDFOLD
      CASE 52
         ;FOLD SPS_TRIG52{H}
         ;ENDFOLD
      CASE 53
         ;FOLD SPS_TRIG53{H}
         ;ENDFOLD
      CASE 54
         ;FOLD SPS_TRIG54{H}
         ;ENDFOLD
      CASE 55
         ;FOLD SPS_TRIG55{H}
         ;ENDFOLD
      CASE 56
         ;FOLD SPS_TRIG56{H}
         ;ENDFOLD
      CASE 57
         ;FOLD SPS_TRIG57{H}
         ;ENDFOLD
      CASE 58
         ;FOLD SPS_TRIG58{H}
         ;ENDFOLD
      CASE 59
         ;FOLD SPS_TRIG59{H}
         ;ENDFOLD
      CASE 60
         ;FOLD SPS_TRIG60{H}
         ;ENDFOLD
      CASE 61
         ;FOLD SPS_TRIG61{H}
         ;ENDFOLD
      CASE 62
         ;FOLD SPS_TRIG62{H}
         ;ENDFOLD
      CASE 63
         ;FOLD SPS_TRIG63{H}
         ;ENDFOLD
      CASE 64
         ;FOLD SPS_TRIG64{H}
         ;ENDFOLD
      CASE 65
         ;FOLD SPS_TRIG65{H}
         ;ENDFOLD
      CASE 66
         ;FOLD SPS_TRIG66{H}
         ;ENDFOLD
      CASE 67
         ;FOLD SPS_TRIG67{H}
         ;ENDFOLD
      CASE 68
         ;FOLD SPS_TRIG68{H}
         ;ENDFOLD
      CASE 69
         ;FOLD SPS_TRIG69{H}
         ;ENDFOLD
      CASE 70
         ;FOLD SPS_TRIG70{H}
         ;ENDFOLD
      CASE 71
         ;FOLD SPS_TRIG71{H}
         ;ENDFOLD
      CASE 72
         ;FOLD SPS_TRIG72{H}
         ;ENDFOLD
      CASE 73
         ;FOLD SPS_TRIG73{H}
         ;ENDFOLD
      CASE 74
         ;FOLD SPS_TRIG74{H}
         ;ENDFOLD
      CASE 75
         ;FOLD SPS_TRIG75{H}
         ;ENDFOLD
      CASE 76
         ;FOLD SPS_TRIG76{H}
         ;ENDFOLD
      CASE 77
         ;FOLD SPS_TRIG77{H}
         ;ENDFOLD
      CASE 78
         ;FOLD SPS_TRIG78{H}
         ;ENDFOLD
      CASE 79
         ;FOLD SPS_TRIG79{H}
         ;ENDFOLD
      CASE 80
         ;FOLD SPS_TRIG80{H}
         ;ENDFOLD
      CASE 81
         ;FOLD SPS_TRIG81{H}
         ;ENDFOLD
      CASE 82
         ;FOLD SPS_TRIG82{H}
         ;ENDFOLD
      CASE 83
         ;FOLD SPS_TRIG83{H}
         ;ENDFOLD
      CASE 84
         ;FOLD SPS_TRIG84{H}
         ;ENDFOLD
      CASE 85
         ;FOLD SPS_TRIG85{H}
         ;ENDFOLD
      CASE 86
         ;FOLD SPS_TRIG86{H}
         ;ENDFOLD
      CASE 87
         ;FOLD SPS_TRIG87{H}
         ;ENDFOLD
      CASE 88
         ;FOLD SPS_TRIG88{H}
         ;ENDFOLD
      CASE 89
         ;FOLD SPS_TRIG89{H}
         ;ENDFOLD
      CASE 90
         ;FOLD SPS_TRIG90{H}
         ;ENDFOLD
      CASE 91
         ;FOLD SPS_TRIG91{H}
         ;ENDFOLD
      CASE 92
         ;FOLD SPS_TRIG92{H}
         ;ENDFOLD
      CASE 93
         ;FOLD SPS_TRIG93{H}
         ;ENDFOLD
      CASE 94
         ;FOLD SPS_TRIG94{H}
         ;ENDFOLD
      CASE 95
         ;FOLD SPS_TRIG95{H}
         ;ENDFOLD
      CASE 96
         ;FOLD SPS_TRIG96{H}
         ;ENDFOLD
      CASE 97
         ;FOLD SPS_TRIG97{H}
         ;ENDFOLD
      CASE 98
         ;FOLD SPS_TRIG98{H}
         ;ENDFOLD
      CASE 99
         ;FOLD SPS_TRIG99{H}
         ;ENDFOLD
      CASE 100
         ;FOLD SPS_TRIG100{H}
         ;ENDFOLD
      CASE 101
         ;FOLD SPS_TRIG101{H}
         ;ENDFOLD
      CASE 102
         ;FOLD SPS_TRIG102{H}
         ;ENDFOLD
      CASE 103
         ;FOLD SPS_TRIG103{H}
         ;ENDFOLD
      CASE 104
         ;FOLD SPS_TRIG104{H}
         ;ENDFOLD
      CASE 105
         ;FOLD SPS_TRIG105{H}
         ;ENDFOLD
      CASE 106
         ;FOLD SPS_TRIG106{H}
         ;ENDFOLD
      CASE 107
         ;FOLD SPS_TRIG107{H}
         ;ENDFOLD
      CASE 108
         ;FOLD SPS_TRIG108{H}
         ;ENDFOLD
      CASE 109
         ;FOLD SPS_TRIG109{H}
         ;ENDFOLD
      CASE 110
         ;FOLD SPS_TRIG110{H}
         ;ENDFOLD
      CASE 111
         ;FOLD SPS_TRIG111{H}
         ;ENDFOLD
      CASE 112
         ;FOLD SPS_TRIG112{H}
         ;ENDFOLD
      CASE 113
         ;FOLD SPS_TRIG113{H}
         ;ENDFOLD
      CASE 114
         ;FOLD SPS_TRIG114{H}
         ;ENDFOLD
   DEFAULT
   ENDSWITCH
   ; FOLD ;%{H}
   IF ($MODE_OP<>#EX) THEN
      ;-- Trigger erst nach Wiederanstart geschaltet --
      IF ((((VW_STOP B_AND 'B10010') >0) AND ((VW_STOP B_AND 'B0001')<=0))) THEN
         ;-- MStep Bewegung --
         HALT
      ENDIF
   ENDIF
   ; ENDFOLD
   IF NOT UES THEN
      SPS_FERTIG=TRUE
   ENDIF
END
; ENDFOLD

--- up24.dat ---
&ACCESS RV7
&REL 180
&COMMENT VW380 Ablegen AFO 115440
&PARAM DISKPATH = KRC:\R1\UPs
&PARAM TEMPLATE = C:\KRC\Roboter\Template\upvorgabe
&PARAM TPVW_VERSION = 8.1.8
&PARAM EDITMASK = Up999[1-999]
DEFDAT  up24
; FOLD ;%{H} %MKUKATPVW
; ENDFOLD
; interface to basic routines
EXT  BAS (BAS_COMMAND  :IN,REAL  :IN )
; interface to VW-standard routines
EXT  VW (VW_COMMAND  :IN,BOOL  :IN,REAL  :IN,REAL  :IN,REAL  :IN,REAL  :IN,BOOL  :IN,E6POS  :IN )
; interface to VW_USER - Call
EXT  VW_USER (VW_USER_CMD  :IN,INT  :IN,REAL  :IN,REAL  :IN,REAL  :IN,REAL  :IN,REAL  :IN,REAL  :IN,BOOL  :IN )
EXT  VW_USR_R (VW_USER_CMD  :IN,INT  :IN,REAL  :IN,REAL  :IN,REAL  :IN,REAL  :IN,REAL  :IN,REAL  :IN,BOOL  :IN )
EXT  IBGN (IBGN_COMMAND  :IN,BOOL  :IN,REAL  :IN,REAL  :IN,BOOL  :IN,E6POS  :OUT )
; interface select routine
EXTFCT  INT  SELECT(SUBTYPE  :IN,INT  :IN,BOOL  :IN,ARI_TYP  :IN,INT  :IN,BOOL_TYP  :IN,INT  :IN,BOOL  :IN)
INT VW_NEXT_FREE=14
INT VW_NFREE_SPS=14
INT VW_MAX_SPS=114
DECL VW_MPARA_TYP P1_D={TOOL_NO 12,BASE_NO 0,VB 100,VE 0,ACC 100,TRG_TIME 0,MOVE_TYPE #PTP_MOTION}
DECL E6POS P1={X 1644.43604,Y -174.747894,Z 2340.60889,A 0.00983779225,B 30.000351,C -90.3522263,S 2,T 42,E1 0.0,E2 0.0,E3 0.0,E4 0.0,E5 0.0,E6 0.0}
DECL VW_MPARA_TYP P2_D={TOOL_NO 12,BASE_NO 0,VB 100,VE 100,ACC 100,TRG_TIME 0,MOVE_TYPE #PTP_MOTION}
DECL E6POS P2={X 1267.49194,Y 829.015381,Z 2086.66602,A 22.4011402,B 19.0144806,C -179.990997,S 2,T 11,E1 0.0,E2 0.0,E3 0.0,E4 0.0,E5 0.0,E6 0.0}
DECL VW_MPARA_TYP P3_D={TOOL_NO 12,BASE_NO 0,VB 100,VE 100,ACC 100,TRG_TIME 0,MOVE_TYPE #PTP_MOTION}
DECL E6POS P3={X -883.151672,Y 1349.00195,Z 2239.81201,A 113.223602,B 15.4502897,C 179.806198,S 2,T 11,E1 0.0,E2 0.0,E3 0.0,E4 0.0,E5 0.0,E6 0.0}
DECL VW_MPARA_TYP P4_D={TOOL_NO 12,BASE_NO 0,VB 100,VE 100,ACC 100,TRG_TIME 0,MOVE_TYPE #PTP_MOTION}
DECL E6POS P4={X -1548.47498,Y 1079.64099,Z 455.632111,A -148.278595,B 89.6800995,C -57.6764984,S 2,T 43,E1 0.0,E2 0.0,E3 0.0,E4 0.0,E5 0.0,E6 0.0}
DECL VW_MPARA_TYP P5_D={TOOL_NO 12,BASE_NO 0,VB 100,VE 100,ACC 100,TRG_TIME 0,MOVE_TYPE #PTP_MOTION}
DECL E6POS P5={X -1548.47498,Y 1079.64099,Z 343.032104,A -148.278595,B 89.6800995,C -57.6764984,S 2,T 43,E1 0.0,E2 0.0,E3 0.0,E4 0.0,E5 0.0,E6 0.0}
DECL VW_MPARA_TYP P6_D={TOOL_NO 12,BASE_NO 0,VB 100,VE 10,ACC 100,TRG_TIME 0,MOVE_TYPE #PTP_MOTION}
DECL E6POS P6={X -1549.21704,Y 1098.57703,Z 143.535202,A -148.278595,B 89.6800995,C -57.6764984,S 2,T 43,E1 0.0,E2 0.0,E3 0.0,E4 0.0,E5 0.0,E6 0.0}
DECL VW_MPARA_TYP P7_D={TOOL_NO 12,BASE_NO 0,VB 250,VE 0,ACC 100,TRG_TIME 5,MOVE_TYPE #PATH_MOTION}
DECL E6POS P7={X -1549.68298,Y 1098.50903,Z 43.2420311,A -179.603806,B 89.8289795,C -89.0018768,S 2,T 43,E1 0.0,E2 0.0,E3 0.0,E4 0.0,E5 0.0,E6 0.0}
DECL VW_MPARA_TYP P8_D={TOOL_NO 12,BASE_NO 0,VB 300,VE 100,ACC 100,TRG_TIME 0,MOVE_TYPE #PATH_MOTION}
DECL E6POS P8={X -1549.21704,Y 1098.57703,Z 143.535004,A -148.277298,B 89.6800766,C -57.6752281,S 2,T 43,E1 0.0,E2 0.0,E3 0.0,E4 0.0,E5 0.0,E6 0.0}
DECL VW_MPARA_TYP P9_D={TOOL_NO 12,BASE_NO 0,VB 100,VE 100,ACC 100,TRG_TIME 0,MOVE_TYPE #PTP_MOTION}
DECL E6POS P9={X -1549.21704,Y 1098.57898,Z 491.046387,A -148.289902,B 89.6801529,C -57.6876411,S 2,T 43,E1 0.0,E2 0.0,E3 0.0,E4 0.0,E5 0.0,E6 0.0}
DECL VW_MPARA_TYP P10_D={TOOL_NO 12,BASE_NO 0,VB 100,VE 100,ACC 100,TRG_TIME 0,MOVE_TYPE #PTP_MOTION}
DECL E6POS P10={X -883.151672,Y 1349.00195,Z 2239.81201,A 113.223602,B 15.4502897,C 179.806198,S 2,T 11,E1 0.0,E2 0.0,E3 0.0,E4 0.0,E5 0.0,E6 0.0}
DECL VW_MPARA_TYP P11_D={TOOL_NO 12,BASE_NO 0,VB 100,VE 100,ACC 100,TRG_TIME 0,MOVE_TYPE #PTP_MOTION}
DECL E6POS P11={X 928.075684,Y 1160.86206,Z 2290.53198,A 40.1389999,B 12.0272198,C 179.585297,S 2,T 11,E1 0.0,E2 0.0,E3 0.0,E4 0.0,E5 0.0,E6 0.0}
DECL VW_MPARA_TYP P12_D={TOOL_NO 12,BASE_NO 0,VB 100,VE 100,ACC 100,TRG_TIME 0,MOVE_TYPE #PTP_MOTION}
DECL E6POS P12={X 1699.01794,Y -188.522598,Z 2233.20703,A -0.975307584,B 34.2327385,C -95.8365479,S 2,T 42,E1 0.0,E2 0.0,E3 0.0,E4 0.0,E5 0.0,E6 0.0}
DECL VW_MPARA_TYP P13_D={TOOL_NO 12,BASE_NO 0,VB 100,VE 0,ACC 100,TRG_TIME 0,MOVE_TYPE #PTP_MOTION}
DECL E6POS P13={X 1644.43604,Y -174.747894,Z 2340.60889,A 0.00983779225,B 30.000351,C -90.3522263,S 2,T 42,E1 0.0,E2 0.0,E3 0.0,E4 0.0,E5 0.0,E6 0.0}
ENDDAT
